// TIA Portal V20 export
TYPE "typeSequenceControlNodetransferPnPLeftJobInterface_GRnR"
// stored: Namespace Unit1.Em5
   STRUCT
      sideTapePICKJob2 : "LER_typeJobInterface";
      hipotThicknessPLACEJob3 : "LER_typeJobInterface";
      hipotThicknessPICKJob4 : "LER_typeJobInterface";
   END_STRUCT;
END_TYPE
